FUNCTION_BLOCK ScrollFS (* Scroll list position engine — accepts ScrollObjectPool_S struct, drives list and scrollbar via Q_ChildPosition *)
  (* Standard: ISO 11783-6; Description: Copyright (c) 2026 Meisterschulen am Ostbahnhof This program and the accompanying materials are made available under the terms of the Eclipse Public License 2.0 which is available at https://www.eclipse.org/legal/epl-2.0/ SPDX-License-Identifier: EPL-2.0 Wraps RampLimitFS (position state, 0..stObj.i32PosMax) and two Q_ChildPosition instances (ISO 11783-6 F.16) that move the list content container and the scrollbar indicator content container. stObj is snapshotted once at INIT via F_MOVE, matching the Q_NumericValue_PHYS pattern. The two Y-position formulas are plain Functions (F_ScrollListY, F_ScrollBarY) — concretely typed, so no ANY-generic MOVE anchoring is needed between them. Pure position logic only — does not read any physical buttons or input fields, see ScrollFS_PHYS for that. See Workspace_Scroll/SCROLL_KONZEPT.md for the full derivation. *)
  (* Version 1.1, 2026-09-05, Franz Höpfinger, Meisterschulen am Ostbahnhof, Add xScale flag, passed through to the internal MoveList/MoveBar (Q_ChildPosition) *)
  (* Version 1.0, 2026-08-09, Franz Höpfinger, Meisterschulen am Ostbahnhof, initial API and implementation and/or initial documentation *)
  PACKAGE isobus::UT::Q;
  IMPORT isobus::utils::scroll::ScrollObjectPool_S;
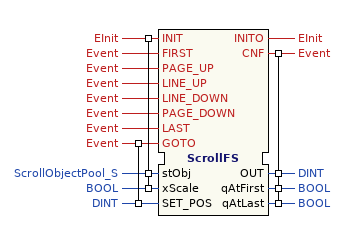
  EVENT_INPUT
    INIT : EInit WITH stObj, xScale; (* Service Initialization *)
    FIRST; (* Jump to the first row (position 0) *)
    PAGE_UP; (* Page up (fast, by stObj.i32Step rows) *)
    LINE_UP; (* One row up *)
    LINE_DOWN; (* One row down *)
    PAGE_DOWN; (* Page down (fast, by stObj.i32Step rows) *)
    LAST; (* Jump to the last row (position stObj.i32PosMax) *)
    GOTO WITH SET_POS; (* Jump to an absolute row position *)
  END_EVENT
  EVENT_OUTPUT
    INITO : EInit; (* Initialization Confirm *)
    CNF WITH OUT, qAtFirst, qAtLast; (* Confirmation of a position change *)
  END_EVENT
  VAR_INPUT
    stObj : isobus::utils::scroll::ScrollObjectPool_S; (* Scroll list object pool properties (list + scrollbar geometry), snapshotted at INIT *)
    xScale : BOOL := FALSE; (* FALSE (default) = bypass, send s16Yposition through unchanged. TRUE = scale it by the DM/SKM factor for the respective parent ID. Passed straight through to the internal MoveList/MoveBar (Q_ChildPosition). *)
    SET_POS : DINT; (* Target position for the GOTO event, clamped to 0..stObj.i32PosMax *)
  END_VAR
  VAR_OUTPUT
    OUT : DINT; (* Current scroll position (0..stObj.i32PosMax, in rows) *)
    qAtFirst : BOOL; (* TRUE if OUT is at row 0 (FIRST reached) - straight passthrough of Ramp.qAtZero *)
    qAtLast : BOOL; (* TRUE if OUT is at row stObj.i32PosMax (LAST reached) - straight passthrough of Ramp.qAtFull *)
  END_VAR
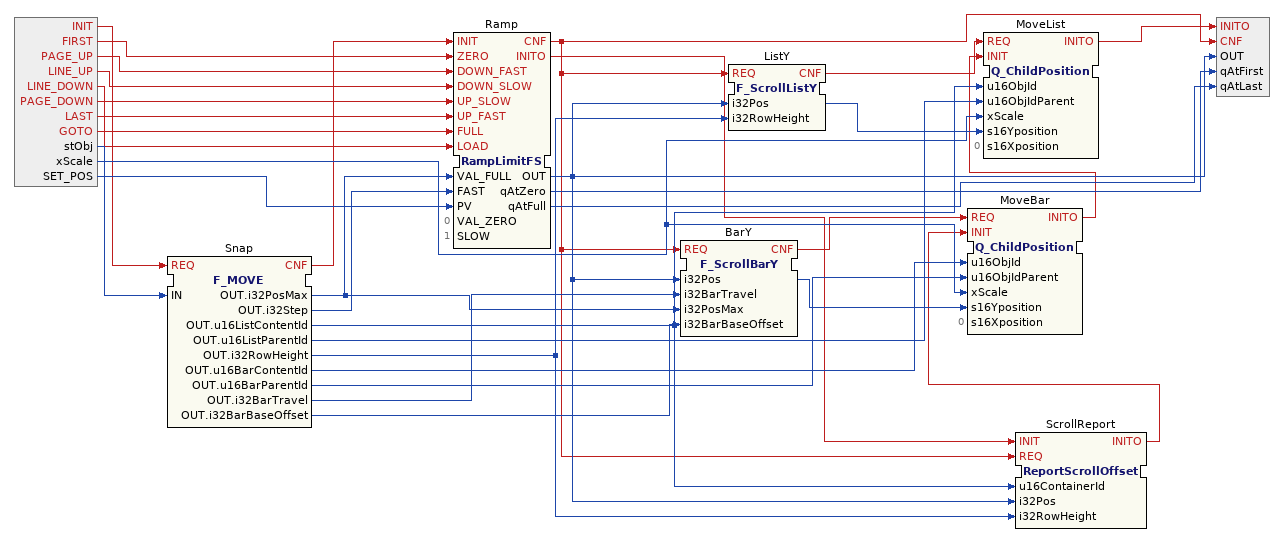
  FBS
    Snap : iec61131::selection::F_MOVE; {SET_ATTRIBUTE(DataType, isobus::utils::scroll::ScrollObjectPool_S)}
    Ramp : eclipse4diac::signalprocessing::RampLimitFS(VAL_ZERO := 0, SLOW := 1);
    MoveList : isobus::UT::Q::Q_ChildPosition(s16Xposition := 0);
    ListY : isobus::UT::Q::helpers::F_ScrollListY;
    MoveBar : isobus::UT::Q::Q_ChildPosition(s16Xposition := 0);
    BarY : isobus::UT::Q::helpers::F_ScrollBarY;
    ScrollReport : isobus::UT::Q::helpers::ReportScrollOffset;
  END_FBS
  EVENT_CONNECTIONS
    INIT TO Snap.REQ;
    Snap.CNF TO Ramp.INIT;
    FIRST TO Ramp.ZERO;
    PAGE_UP TO Ramp.DOWN_FAST;
    LINE_UP TO Ramp.DOWN_SLOW;
    LINE_DOWN TO Ramp.UP_SLOW;
    PAGE_DOWN TO Ramp.UP_FAST;
    LAST TO Ramp.FULL;
    GOTO TO Ramp.LOAD;
    Ramp.CNF TO CNF;
    Ramp.CNF TO ListY.REQ;
    ListY.CNF TO MoveList.REQ;
    Ramp.CNF TO BarY.REQ;
    BarY.CNF TO MoveBar.REQ;
    Ramp.INITO TO ScrollReport.INIT;
    Ramp.CNF TO ScrollReport.REQ;
    ScrollReport.INITO TO MoveBar.INIT;
    MoveBar.INITO TO MoveList.INIT;
    MoveList.INITO TO INITO;
  END_CONNECTIONS
  DATA_CONNECTIONS
    stObj TO Snap.IN;
    Snap.OUT.i32PosMax TO Ramp.VAL_FULL;
    Snap.OUT.i32Step TO Ramp.FAST;
    SET_POS TO Ramp.PV;
    Ramp.OUT TO OUT;
    Ramp.qAtZero TO qAtFirst;
    Ramp.qAtFull TO qAtLast;
    Snap.OUT.u16ListContentId TO MoveList.u16ObjId;
    Snap.OUT.u16ListParentId TO MoveList.u16ObjIdParent;
    xScale TO MoveList.xScale;
    Ramp.OUT TO ListY.i32Pos;
    Snap.OUT.i32RowHeight TO ListY.i32RowHeight;
    ListY. TO MoveList.s16Yposition;
    Snap.OUT.u16BarContentId TO MoveBar.u16ObjId;
    Snap.OUT.u16BarParentId TO MoveBar.u16ObjIdParent;
    xScale TO MoveBar.xScale;
    Ramp.OUT TO BarY.i32Pos;
    Snap.OUT.i32BarTravel TO BarY.i32BarTravel;
    Snap.OUT.i32PosMax TO BarY.i32PosMax;
    Snap.OUT.i32BarBaseOffset TO BarY.i32BarBaseOffset;
    BarY. TO MoveBar.s16Yposition;
    Snap.OUT.u16ListContentId TO ScrollReport.u16ContainerId;
    Ramp.OUT TO ScrollReport.i32Pos;
    Snap.OUT.i32RowHeight TO ScrollReport.i32RowHeight;
  END_CONNECTIONS
END_FUNCTION_BLOCK
